LIN {X 0,Y 81.103,Z 363.12,A -85,B 0,C 180,E1 -27834.313,E2 -27834.313} C_VEL
LIN {X 0,Y 82.768,Z 358.459,A -85,B 0,C 180,E1 -27837.848,E2 -27837.848} C_VEL
LIN {X 0,Y 84.322,Z 351.512,A -85,B 0,C 180,E1 -27842.351,E2 -27842.351} C_VEL
LIN {X 0,Y 85.789,Z 343.802,A -85,B 0,C 180,E1 -27846.444,E2 -27846.444} C_VEL
LIN {X 0,Y 86.709,Z 336.677,A -85,B 0,C 180,E1 -27849.672,E2 -27849.672} C_VEL
LIN {X 0,Y 87.275,Z 327.984,A -85,B 0,C 180,E1 -27853.08,E2 -27853.08} C_VEL
LIN {X 0,Y 87.272,Z 324.602,A -85,B 0,C 180,E1 -27854.371,E2 -27854.371} C_VEL
LIN {X 0,Y 84.695,Z 316.637,A -85,B 0,C 180,E1 -27858.324,E2 -27858.324} C_VEL
LIN {X 0,Y 82.109,Z 312.261,A -85,B 0,C 180,E1 -27861.198,E2 -27861.198} C_VEL
LIN {X 0,Y 79.987,Z 309.343,A -85,B 0,C 180,E1 -27863.483,E2 -27863.483} C_VEL
LIN {X 0,Y 79.503,Z 307.393,A -85,B 0,C 180,E1 -27864.498,E2 -27864.498} C_VEL
LIN {X 0,Y 79.529,Z 307.39,A -85,B 0,C 180,E1 -27873.768,E2 -27873.768} C_VEL
LIN {X 0,Y 79.498,Z 307.382,A -85,B 0,C 180,E1 -27879.282,E2 -27879.282} C_VEL
LIN {X 0,Y 79.799,Z 307.348,A -85,B 0,C 180,E1 -27885.672,E2 -27885.672} C_VEL
LIN {X 0,Y 79.947,Z 307.327,A -85,B 0,C 180,E1 -27889.865,E2 -27889.865} C_VEL
LIN {X 0,Y 80.641,Z 307.236,A -85,B 0,C 180,E1 -27899.991,E2 -27899.991} C_VEL
LIN {X 0,Y 80,Z 307.314,A -85,B 0,C 180,E1 -27910.11,E2 -27910.11} C_VEL
LIN {X 0,Y 79.768,Z 307.361,A -85,B 0,C 180,E1 -27915.317,E2 -27915.317} C_VEL
LIN {X 0,Y 79.517,Z 307.376,A -85,B 0,C 180,E1 -27920.693,E2 -27920.693} C_VEL
LIN {X 0,Y 79.487,Z 307.396,A -85,B 0,C 180,E1 -27927.837,E2 -27927.837} C_VEL
LIN {X 0,Y 79.465,Z 307.398,A -85,B 0,C 180,E1 -27937.243,E2 -27937.243} C_VEL
LIN {X 0,Y 79.492,Z 307.392,A -85,B 0,C 180,E1 -27945.001,E2 -27945.001} C_VEL
LIN {X 0,Y 79.475,Z 307.522,A -85,B 0,C 180,E1 -27951.107,E2 -27951.107} C_VEL
LIN {X 0,Y 80.071,Z 309.557,A -85,B 0,C 180,E1 -27952.164,E2 -27952.164} C_VEL
LIN {X 0,Y 81.96,Z 312.404,A -85,B 0,C 180,E1 -27954.533,E2 -27954.533} C_VEL
LIN {X 0,Y 84.975,Z 318.525,A -85,B 0,C 180,E1 -27958.565,E2 -27958.565} C_VEL
LIN {X 0,Y 87.806,Z 325.654,A -85,B 0,C 180,E1 -27962.905,E2 -27962.905} C_VEL
LIN {X 0,Y 89.004,Z 331.434,A -85,B 0,C 180,E1 -27966.098,E2 -27966.098} C_VEL
LIN {X 0,Y 88.877,Z 336.304,A -85,B 0,C 180,E1 -27968.542,E2 -27968.542} C_VEL
LIN {X 0,Y 88.422,Z 338.689,A -85,B 0,C 180,E1 -27969.645,E2 -27969.645} C_VEL
LIN {X 0,Y 84.98,Z 348.04,A -85,B 0,C 180,E1 -27974.402,E2 -27974.402} C_VEL
LIN {X 0,Y 82.427,Z 354.664,A -85,B 0,C 180,E1 -27978.933,E2 -27978.933} C_VEL
LIN {X 0,Y 80.368,Z 360.174,A -85,B 0,C 180,E1 -27983.718,E2 -27983.718} C_VEL
LIN {X 0,Y 78.415,Z 365.767,A -85,B 0,C 180,E1 -27989.993,E2 -27989.993} C_VEL
LIN {X 0,Y 78.325,Z 366.053,A -85,B 0,C 180,E1 -27990.371,E2 -27990.371} C_VEL
LIN {X 0,Y 76.885,Z 368.828,A -85,B 0,C 180,E1 -27994.107,E2 -27994.107} C_VEL
LIN {X 0,Y 73.232,Z 372.559,A -85,B 0,C 180,E1 -28000.555,E2 -28000.555} C_VEL
LIN {X 0,Y 70.419,Z 375.498,A -85,B 0,C 180,E1 -28007.834,E2 -28007.834} C_VEL
LIN {X 0,Y 70.359,Z 376.852,A -85,B 0,C 180,E1 -28012.526,E2 -28012.526} C_VEL
LIN {X 0,Y 71.985,Z 378.249,A -85,B 0,C 180,E1 -28019.211,E2 -28019.211} C_VEL
LIN {X 0,Y 74.077,Z 378.865,A -85,B 0,C 180,E1 -28024.689,E2 -28024.689} C_VEL
LIN {X 0,Y 76.782,Z 378.987,A -85,B 0,C 180,E1 -28029.837,E2 -28029.837} C_VEL
LIN {X 0,Y 81.363,Z 378.263,A -85,B 0,C 180,E1 -28036.302,E2 -28036.302} C_VEL
LIN {X 0,Y 83.749,Z 377.668,A -85,B 0,C 180,E1 -28039.038,E2 -28039.038} C_VEL
LIN {X 0,Y 90.093,Z 375.178,A -85,B 0,C 180,E1 -28044.982,E2 -28044.982} C_VEL
LIN {X 0,Y 97.253,Z 371.306,A -85,B 0,C 180,E1 -28050.121,E2 -28050.121} C_VEL
LIN {X 0,Y 99.807,Z 369.765,A -85,B 0,C 180,E1 -28051.654,E2 -28051.654} C_VEL
LIN {X 0,Y 101.693,Z 367.889,A -85,B 0,C 180,E1 -28053.94,E2 -28053.94} C_VEL
LIN {X 0,Y 102.888,Z 365.535,A -85,B 0,C 180,E1 -28057.941,E2 -28057.941} C_VEL
LIN {X 0,Y 103.573,Z 363.322,A -85,B 0,C 180,E1 -28061.783,E2 -28061.783} C_VEL
LIN {X 0,Y 103.925,Z 362.042,A -85,B 0,C 180,E1 -28064.313,E2 -28064.313} C_VEL
LIN {X 0,Y 104.24,Z 360.271,A -85,B 0,C 180,E1 -28068.338,E2 -28068.338} C_VEL
LIN {X 0,Y 104.447,Z 358.742,A -85,B 0,C 180,E1 -28072.273,E2 -28072.273} C_VEL
LIN {X 0,Y 105.03,Z 356.721,A -85,B 0,C 180,E1 -28080.007,E2 -28080.007} C_VEL
LIN {X 0,Y 105.33,Z 356.2,A -85,B 0,C 180,E1 -28083.833,E2 -28083.833} C_VEL
LIN {X 0,Y 104.851,Z 356.834,A -85,B 0,C 180,E1 -28087.711,E2 -28087.711} C_VEL
LIN {X 0,Y 104.027,Z 359.222,A -85,B 0,C 180,E1 -28095.685,E2 -28095.685} C_VEL
LIN {X 0,Y 103.777,Z 360.902,A -85,B 0,C 180,E1 -28099.799,E2 -28099.799} C_VEL
LIN {X 0,Y 103.283,Z 364.111,A -85,B 0,C 180,E1 -28105.717,E2 -28105.717} C_VEL
LIN {X 0,Y 102.359,Z 367.453,A -85,B 0,C 180,E1 -28111.002,E2 -28111.002} C_VEL
LIN {X 0,Y 101.72,Z 369.604,A -85,B 0,C 180,E1 -28114.004,E2 -28114.004} C_VEL
LIN {X 0,Y 100.581,Z 371.544,A -85,B 0,C 180,E1 -28116.539,E2 -28116.539} C_VEL
LIN {X 0,Y 96.125,Z 375.798,A -85,B 0,C 180,E1 -28121.158,E2 -28121.158} C_VEL
LIN {X 0,Y 92.817,Z 378.218,A -85,B 0,C 180,E1 -28124.01,E2 -28124.01} C_VEL
LIN {X 0,Y 86.169,Z 381.587,A -85,B 0,C 180,E1 -28129.279,E2 -28129.279} C_VEL
LIN {X 0,Y 82.146,Z 383.226,A -85,B 0,C 180,E1 -28133.219,E2 -28133.219} C_VEL
LIN {X 0,Y 78.577,Z 384.271,A -85,B 0,C 180,E1 -28137.552,E2 -28137.552} C_VEL
LIN {X 0,Y 75.641,Z 384.853,A -85,B 0,C 180,E1 -28142.326,E2 -28142.326} C_VEL
LIN {X 0,Y 73.297,Z 385,A -85,B 0,C 180,E1 -28147.455,E2 -28147.455} C_VEL
LIN {X 0,Y 71.542,Z 384.699,A -85,B 0,C 180,E1 -28152.868,E2 -28152.868} C_VEL
LIN {X 0,Y 70.469,Z 383.825,A -85,B 0,C 180,E1 -28158.502,E2 -28158.502} C_VEL
LIN {X 0,Y 70.06,Z 382.441,A -85,B 0,C 180,E1 -28164.25,E2 -28164.25} C_VEL
LIN {X 0,Y 70.143,Z 380.555,A -85,B 0,C 180,E1 -28170.007,E2 -28170.007} C_VEL
LIN {X 0,Y 70.183,Z 376.533,A -85,B 0,C 180,E1 -28178.646,E2 -28178.646} C_VEL
LIN {X 0,Y 70.879,Z 372.999,A -85,B 0,C 180,E1 -28184.36,E2 -28184.36} C_VEL
LIN {X 0,Y 72.632,Z 367.54,A -85,B 0,C 180,E1 -28191.283,E2 -28191.283} C_VEL
LIN {X 0,Y 75.263,Z 360.701,A -85,B 0,C 180,E1 -28197.841,E2 -28197.841} C_VEL
LIN {X 0,Y 77.339,Z 353.736,A -85,B 0,C 180,E1 -28203.049,E2 -28203.049} C_VEL
LIN {X 0,Y 79.321,Z 344.848,A -85,B 0,C 180,E1 -28208.34,E2 -28208.34} C_VEL
LIN {X 0,Y 80.625,Z 336.415,A -85,B 0,C 180,E1 -28212.506,E2 -28212.506} C_VEL
LIN {X 0,Y 81.34,Z 329.032,A -85,B 0,C 180,E1 -28215.661,E2 -28215.661} C_VEL
LIN {X 0,Y 81.384,Z 327.475,A -85,B 0,C 180,E1 -28216.292,E2 -28216.292} C_VEL
LIN {X 0,Y 79.775,Z 321.356,A -85,B 0,C 180,E1 -28219.762,E2 -28219.762} C_VEL
LIN {X 0,Y 75.378,Z 313.535,A -85,B 0,C 180,E1 -28225.974,E2 -28225.974} C_VEL
LIN {X 0,Y 72.881,Z 310.248,A -85,B 0,C 180,E1 -28229.373,E2 -28229.373} C_VEL
LIN {X 0,Y 72.367,Z 308.273,A -85,B 0,C 180,E1 -28230.74,E2 -28230.74} C_VEL
LIN {X 0,Y 72.388,Z 308.265,A -85,B 0,C 180,E1 -28237.138,E2 -28237.138} C_VEL
LIN {X 0,Y 72.69,Z 308.235,A -85,B 0,C 180,E1 -28245.231,E2 -28245.231} C_VEL
LIN {X 0,Y 72.838,Z 308.207,A -85,B 0,C 180,E1 -28248.864,E2 -28248.864} C_VEL
LIN {X 0,Y 73.568,Z 308.116,A -85,B 0,C 180,E1 -28259.99,E2 -28259.99} C_VEL
LIN {X 0,Y 72.886,Z 308.2,A -85,B 0,C 180,E1 -28271.109,E2 -28271.109} C_VEL
LIN {X 0,Y 72.587,Z 308.255,A -85,B 0,C 180,E1 -28276.875,E2 -28276.875} C_VEL
LIN {X 0,Y 72.398,Z 308.262,A -85,B 0,C 180,E1 -28282.837,E2 -28282.837} C_VEL
LIN {X 0,Y 72.378,Z 308.279,A -85,B 0,C 180,E1 -28289.07,E2 -28289.07} C_VEL
LIN {X 0,Y 72.348,Z 308.281,A -85,B 0,C 180,E1 -28295.638,E2 -28295.638} C_VEL
LIN {X 0,Y 72.329,Z 308.288,A -85,B 0,C 180,E1 -28302.842,E2 -28302.842} C_VEL
LIN {X 0,Y 72.465,Z 308.387,A -85,B 0,C 180,E1 -28305.068,E2 -28305.068} C_VEL
LIN {X 0,Y 72.973,Z 310.272,A -85,B 0,C 180,E1 -28306.294,E2 -28306.294} C_VEL
LIN {X 0,Y 75.152,Z 313.541,A -85,B 0,C 180,E1 -28309.756,E2 -28309.756} C_VEL
LIN {X 0,Y 77.952,Z 318.904,A -85,B 0,C 180,E1 -28314.218,E2 -28314.218} C_VEL
LIN {X 0,Y 81.181,Z 326.703,A -85,B 0,C 180,E1 -28319.945,E2 -28319.945} C_VEL
LIN {X 0,Y 82.523,Z 331.958,A -85,B 0,C 180,E1 -28323.382,E2 -28323.382} C_VEL
LIN {X 0,Y 82.753,Z 335.584,A -85,B 0,C 180,E1 -28325.536,E2 -28325.536} C_VEL
LIN {X 0,Y 82.192,Z 339.102,A -85,B 0,C 180,E1 -28327.363,E2 -28327.363} C_VEL
LIN {X 0,Y 78.825,Z 347.551,A -85,B 0,C 180,E1 -28331.81,E2 -28331.81} C_VEL
LIN {X 0,Y 75.411,Z 355.758,A -85,B 0,C 180,E1 -28337.889,E2 -28337.889} C_VEL
LIN {X 0,Y 73.223,Z 361.141,A -85,B 0,C 180,E1 -28343.102,E2 -28343.102} C_VEL
LIN {X 0,Y 71.344,Z 366.236,A -85,B 0,C 180,E1 -28349.444,E2 -28349.444} C_VEL
LIN {X 0,Y 70.153,Z 370.18,A -85,B 0,C 180,E1 -28355.742,E2 -28355.742} C_VEL
LIN {X 0,Y 69.606,Z 374.297,A -85,B 0,C 180,E1 -28364.613,E2 -28364.613} C_VEL
LIN {X 0,Y 70.359,Z 376.852,A -85,B 0,C 180,E1 -28372.526,E2 -28372.526} C_VEL
LIN {X 0,Y 70.741,Z 377.994,A -85,B 0,C 180,E1 -28377.215,E2 -28377.215} C_VEL
LIN {X 0,Y 70.592,Z 379.038,A -85,B 0,C 180,E1 -28385.209,E2 -28385.209} C_VEL
LIN {X 0,Y 71.757,Z 379.279,A -85,B 0,C 180,E1 -28393.169,E2 -28393.169} C_VEL
LIN {X 0,Y 74.073,Z 378.93,A -85,B 0,C 180,E1 -28397.453,E2 -28397.453} C_VEL
LIN {X 0,Y 79.102,Z 377.841,A -85,B 0,C 180,E1 -28403.083,E2 -28403.083} C_VEL
LIN {X 0,Y 86.063,Z 375.201,A -85,B 0,C 180,E1 -28409.018,E2 -28409.018} C_VEL
LIN {X 0,Y 91.133,Z 372.776,A -85,B 0,C 180,E1 -28412.448,E2 -28412.448} C_VEL
LIN {X 0,Y 93.808,Z 371.228,A -85,B 0,C 180,E1 -28414.017,E2 -28414.017} C_VEL
LIN {X 0,Y 95.899,Z 369.544,A -85,B 0,C 180,E1 -28416.583,E2 -28416.583} C_VEL
LIN {X 0,Y 96.958,Z 367.597,A -85,B 0,C 180,E1 -28420.425,E2 -28420.425} C_VEL
LIN {X 0,Y 97.577,Z 366.357,A -85,B 0,C 180,E1 -28423.264,E2 -28423.264} C_VEL
LIN {X 0,Y 98.135,Z 364.597,A -85,B 0,C 180,E1 -28427.601,E2 -28427.601} C_VEL
LIN {X 0,Y 98.601,Z 363.162,A -85,B 0,C 180,E1 -28431.812,E2 -28431.812} C_VEL
LIN {X 0,Y 98.977,Z 362.135,A -85,B 0,C 180,E1 -28435.936,E2 -28435.936} C_VEL
LIN {X 0,Y 99.472,Z 361.225,A -85,B 0,C 180,E1 -28440.007,E2 -28440.007} C_VEL
LIN {X 0,Y 99.771,Z 360.797,A -85,B 0,C 180,E1 -28444.047,E2 -28444.047} C_VEL
LIN {X 0,Y 99.209,Z 361.498,A -85,B 0,C 180,E1 -28448.152,E2 -28448.152} C_VEL
LIN {X 0,Y 98.286,Z 363.955,A -85,B 0,C 180,E1 -28456.627,E2 -28456.627} C_VEL
LIN {X 0,Y 97.745,Z 365.713,A -85,B 0,C 180,E1 -28461.077,E2 -28461.077} C_VEL
LIN {X 0,Y 97.072,Z 368.008,A -85,B 0,C 180,E1 -28465.755,E2 -28465.755} C_VEL
LIN {X 0,Y 95.885,Z 370.907,A -85,B 0,C 180,E1 -28470.877,E2 -28470.877} C_VEL
LIN {X 0,Y 95.224,Z 372.222,A -85,B 0,C 180,E1 -28473.072,E2 -28473.072} C_VEL
LIN {X 0,Y 94.194,Z 373.557,A -85,B 0,C 180,E1 -28474.852,E2 -28474.852} C_VEL
LIN {X 0,Y 90.193,Z 376.729,A -85,B 0,C 180,E1 -28478.821,E2 -28478.821} C_VEL
LIN {X 0,Y 87.979,Z 378.178,A -85,B 0,C 180,E1 -28480.644,E2 -28480.644} C_VEL
LIN {X 0,Y 80.906,Z 381.44,A -85,B 0,C 180,E1 -28485.988,E2 -28485.988} C_VEL
LIN {X 0,Y 76.576,Z 383.034,A -85,B 0,C 180,E1 -28490.035,E2 -28490.035} C_VEL
LIN {X 0,Y 72.682,Z 384.05,A -85,B 0,C 180,E1 -28494.547,E2 -28494.547} C_VEL
LIN {X 0,Y 69.407,Z 384.559,A -85,B 0,C 180,E1 -28499.592,E2 -28499.592} C_VEL
LIN {X 0,Y 66.773,Z 384.631,A -85,B 0,C 180,E1 -28505.111,E2 -28505.111} C_VEL
LIN {X 0,Y 64.779,Z 384.266,A -85,B 0,C 180,E1 -28511.014,E2 -28511.014} C_VEL
LIN {X 0,Y 63.527,Z 383.382,A -85,B 0,C 180,E1 -28517.225,E2 -28517.225} C_VEL
LIN {X 0,Y 63.022,Z 381.928,A -85,B 0,C 180,E1 -28523.606,E2 -28523.606} C_VEL
LIN {X 0,Y 63.059,Z 379.963,A -85,B 0,C 180,E1 -28530.008,E2 -28530.008} C_VEL
LIN {X 0,Y 62.99,Z 377.38,A -85,B 0,C 180,E1 -28536.414,E2 -28536.414} C_VEL
LIN {X 0,Y 63.997,Z 372.229,A -85,B 0,C 180,E1 -28545.943,E2 -28545.943} C_VEL
LIN {X 0,Y 66.032,Z 366.67,A -85,B 0,C 180,E1 -28553.532,E2 -28553.532} C_VEL
LIN {X 0,Y 68.998,Z 359.659,A -85,B 0,C 180,E1 -28560.625,E2 -28560.625} C_VEL
LIN {X 0,Y 71.216,Z 352.438,A -85,B 0,C 180,E1 -28566.316,E2 -28566.316} C_VEL
LIN {X 0,Y 73.153,Z 345.059,A -85,B 0,C 180,E1 -28571.024,E2 -28571.024} C_VEL
LIN {X 0,Y 74.688,Z 336.867,A -85,B 0,C 180,E1 -28575.436,E2 -28575.436} C_VEL
LIN {X 0,Y 75.561,Z 329.807,A -85,B 0,C 180,E1 -28578.792,E2 -28578.792} C_VEL
LIN {X 0,Y 74.909,Z 326.782,A -85,B 0,C 180,E1 -28580.695,E2 -28580.695} C_VEL
LIN {X 0,Y 72.798,Z 322.258,A -85,B 0,C 180,E1 -28584.591,E2 -28584.591} C_VEL
LIN {X 0,Y 70.569,Z 318.168,A -85,B 0,C 180,E1 -28588.465,E2 -28588.465} C_VEL
LIN {X 0,Y 68.016,Z 313.925,A -85,B 0,C 180,E1 -28593.379,E2 -28593.379} C_VEL
LIN {X 0,Y 66.142,Z 311.65,A -85,B 0,C 180,E1 -28596.921,E2 -28596.921} C_VEL
LIN {X 0,Y 65.314,Z 309.148,A -85,B 0,C 180,E1 -28599.519,E2 -28599.519} C_VEL
LIN {X 0,Y 65.732,Z 309.091,A -85,B 0,C 180,E1 -28607.642,E2 -28607.642} C_VEL
LIN {X 0,Y 66.466,Z 309,A -85,B 0,C 180,E1 -28619.989,E2 -28619.989} C_VEL
LIN {X 0,Y 65.942,Z 309.081,A -85,B 0,C 180,E1 -28626.107,E2 -28626.107} C_VEL
LIN {X 0,Y 65.779,Z 309.088,A -85,B 0,C 180,E1 -28632.327,E2 -28632.327} C_VEL
LIN {X 0,Y 65.39,Z 309.144,A -85,B 0,C 180,E1 -28638.798,E2 -28638.798} C_VEL
LIN {X 0,Y 65.25,Z 309.165,A -85,B 0,C 180,E1 -28645.508,E2 -28645.508} C_VEL
LIN {X 0,Y 65.221,Z 309.174,A -85,B 0,C 180,E1 -28652.587,E2 -28652.587} C_VEL
LIN {X 0,Y 65.334,Z 309.367,A -85,B 0,C 180,E1 -28656.259,E2 -28656.259} C_VEL
LIN {X 0,Y 65.799,Z 311.001,A -85,B 0,C 180,E1 -28657.876,E2 -28657.876} C_VEL
LIN {X 0,Y 67.783,Z 313.741,A -85,B 0,C 180,E1 -28662.229,E2 -28662.229} C_VEL
LIN {X 0,Y 70.259,Z 317.764,A -85,B 0,C 180,E1 -28667.066,E2 -28667.066} C_VEL
LIN {X 0,Y 72.915,Z 323.466,A -85,B 0,C 180,E1 -28672.657,E2 -28672.657} C_VEL
LIN {X 0,Y 75.017,Z 329.123,A -85,B 0,C 180,E1 -28677.457,E2 -28677.457} C_VEL
LIN {X 0,Y 76.285,Z 333.805,A -85,B 0,C 180,E1 -28681.009,E2 -28681.009} C_VEL
LIN {X 0,Y 76.509,Z 337.183,A -85,B 0,C 180,E1 -28683.389,E2 -28683.389} C_VEL
LIN {X 0,Y 76.114,Z 339.515,A -85,B 0,C 180,E1 -28684.712,E2 -28684.712} C_VEL
LIN {X 0,Y 72.108,Z 348.813,A -85,B 0,C 180,E1 -28690.047,E2 -28690.047} C_VEL
LIN {X 0,Y 69.111,Z 355.415,A -85,B 0,C 180,E1 -28695.264,E2 -28695.264} C_VEL
LIN {X 0,Y 66.658,Z 360.911,A -85,B 0,C 180,E1 -28700.893,E2 -28700.893} C_VEL
LIN {X 0,Y 64.705,Z 365.52,A -85,B 0,C 180,E1 -28706.879,E2 -28706.879} C_VEL
LIN {X 0,Y 63.357,Z 369.531,A -85,B 0,C 180,E1 -28713.509,E2 -28713.509} C_VEL
LIN {X 0,Y 62.52,Z 373.752,A -85,B 0,C 180,E1 -28722.984,E2 -28722.984} C_VEL
LIN {X 0,Y 62.803,Z 375.992,A -85,B 0,C 180,E1 -28729.607,E2 -28729.607} C_VEL
LIN {X 0,Y 63.892,Z 377.664,A -85,B 0,C 180,E1 -28736.094,E2 -28736.094} C_VEL
LIN {X 0,Y 65.667,Z 378.723,A -85,B 0,C 180,E1 -28742.342,E2 -28742.342} C_VEL
LIN {X 0,Y 68.155,Z 379.251,A -85,B 0,C 180,E1 -28748.212,E2 -28748.212} C_VEL
LIN {X 0,Y 71.301,Z 379.283,A -85,B 0,C 180,E1 -28753.617,E2 -28753.617} C_VEL
LIN {X 0,Y 74.073,Z 378.93,A -85,B 0,C 180,E1 -28757.453,E2 -28757.453} C_VEL
LIN {X 0,Y 76.749,Z 378.431,A -85,B 0,C 180,E1 -28761.441,E2 -28761.441} C_VEL
LIN {X 0,Y 80.34,Z 376.992,A -85,B 0,C 180,E1 -28768.109,E2 -28768.109} C_VEL
LIN {X 0,Y 84.66,Z 374.573,A -85,B 0,C 180,E1 -28774.095,E2 -28774.095} C_VEL
LIN {X 0,Y 88.275,Z 372.535,A -85,B 0,C 180,E1 -28776.894,E2 -28776.894} C_VEL
LIN {X 0,Y 90.057,Z 371.146,A -85,B 0,C 180,E1 -28779.45,E2 -28779.45} C_VEL
LIN {X 0,Y 90.785,Z 370.22,A -85,B 0,C 180,E1 -28781.97,E2 -28781.97} C_VEL
LIN {X 0,Y 91.685,Z 368.508,A -85,B 0,C 180,E1 -28786.714,E2 -28786.714} C_VEL
LIN {X 0,Y 92.427,Z 367.193,A -85,B 0,C 180,E1 -28791.261,E2 -28791.261} C_VEL
LIN {X 0,Y 93,Z 366.154,A -85,B 0,C 180,E1 -28795.674,E2 -28795.674} C_VEL
LIN {X 0,Y 93.575,Z 365.328,A -85,B 0,C 180,E1 -28800.008,E2 -28800.008} C_VEL
LIN {X 0,Y 93.902,Z 365.023,A -85,B 0,C 180,E1 -28804.3,E2 -28804.3} C_VEL
LIN {X 0,Y 92.931,Z 366.213,A -85,B 0,C 180,E1 -28810.57,E2 -28810.57} C_VEL
LIN {X 0,Y 92.023,Z 368.332,A -85,B 0,C 180,E1 -28817.795,E2 -28817.795} C_VEL
LIN {X 0,Y 91.252,Z 370.118,A -85,B 0,C 180,E1 -28822.657,E2 -28822.657} C_VEL
LIN {X 0,Y 90.04,Z 372.537,A -85,B 0,C 180,E1 -28827.934,E2 -28827.934} C_VEL
LIN {X 0,Y 89.377,Z 373.689,A -85,B 0,C 180,E1 -28830.134,E2 -28830.134} C_VEL
LIN {X 0,Y 87.87,Z 375.231,A -85,B 0,C 180,E1 -28832.892,E2 -28832.892} C_VEL
LIN {X 0,Y 85.533,Z 376.888,A -85,B 0,C 180,E1 -28835.121,E2 -28835.121} C_VEL
LIN {X 0,Y 83.342,Z 378.166,A -85,B 0,C 180,E1 -28836.953,E2 -28836.953} C_VEL
LIN {X 0,Y 75.947,Z 381.294,A -85,B 0,C 180,E1 -28842.253,E2 -28842.253} C_VEL
LIN {X 0,Y 71.28,Z 382.818,A -85,B 0,C 180,E1 -28846.366,E2 -28846.366} C_VEL
LIN {X 0,Y 67.025,Z 383.824,A -85,B 0,C 180,E1 -28851.024,E2 -28851.024} C_VEL
LIN {X 0,Y 63.365,Z 384.264,A -85,B 0,C 180,E1 -28856.329,E2 -28856.329} C_VEL
LIN {X 0,Y 60.391,Z 384.264,A -85,B 0,C 180,E1 -28862.268,E2 -28862.268} C_VEL
LIN {X 0,Y 58.107,Z 383.825,A -85,B 0,C 180,E1 -28868.735,E2 -28868.735} C_VEL
LIN {X 0,Y 56.614,Z 382.916,A -85,B 0,C 180,E1 -28875.634,E2 -28875.634} C_VEL
LIN {X 0,Y 55.889,Z 380.484,A -85,B 0,C 180,E1 -28886.405,E2 -28886.405} C_VEL
LIN {X 0,Y 55.977,Z 379.372,A -85,B 0,C 180,E1 -28890.009,E2 -28890.009} C_VEL
LIN {X 0,Y 55.933,Z 376.703,A -85,B 0,C 180,E1 -28897.228,E2 -28897.228} C_VEL
LIN {X 0,Y 56.587,Z 373.391,A -85,B 0,C 180,E1 -28904.392,E2 -28904.392} C_VEL
LIN {X 0,Y 58.437,Z 368.164,A -85,B 0,C 180,E1 -28913.018,E2 -28913.018} C_VEL
LIN {X 0,Y 60.784,Z 363.037,A -85,B 0,C 180,E1 -28919.442,E2 -28919.442} C_VEL
LIN {X 0,Y 62.874,Z 358.546,A -85,B 0,C 180,E1 -28923.989,E2 -28923.989} C_VEL
LIN {X 0,Y 65.375,Z 351.116,A -85,B 0,C 180,E1 -28930.177,E2 -28930.177} C_VEL
LIN {X 0,Y 67.453,Z 343.961,A -85,B 0,C 180,E1 -28935.006,E2 -28935.006} C_VEL
LIN {X 0,Y 69.198,Z 336.038,A -85,B 0,C 180,E1 -28939.531,E2 -28939.531} C_VEL
LIN {X 0,Y 69.774,Z 332.099,A -85,B 0,C 180,E1 -28941.678,E2 -28941.678} C_VEL
LIN {X 0,Y 68.903,Z 329.013,A -85,B 0,C 180,E1 -28944.258,E2 -28944.258} C_VEL
LIN {X 0,Y 66.459,Z 323.752,A -85,B 0,C 180,E1 -28949.835,E2 -28949.835} C_VEL
LIN {X 0,Y 64.589,Z 320.325,A -85,B 0,C 180,E1 -28954.188,E2 -28954.188} C_VEL
LIN {X 0,Y 62.717,Z 317.648,A -85,B 0,C 180,E1 -28958.63,E2 -28958.63} C_VEL
LIN {X 0,Y 62.276,Z 316.478,A -85,B 0,C 180,E1 -28960.199,E2 -28960.199} C_VEL
LIN {X 0,Y 61.209,Z 314.774,A -85,B 0,C 180,E1 -28963.548,E2 -28963.548} C_VEL
LIN {X 0,Y 59.096,Z 311.463,A -85,B 0,C 180,E1 -28972.084,E2 -28972.084} C_VEL
LIN {X 0,Y 58.918,Z 309.955,A -85,B 0,C 180,E1 -28974.855,E2 -28974.855} C_VEL
LIN {X 0,Y 59.359,Z 309.884,A -85,B 0,C 180,E1 -28979.988,E2 -28979.988} C_VEL
LIN {X 0,Y 58.825,Z 309.963,A -85,B 0,C 180,E1 -28986.849,E2 -28986.849} C_VEL
LIN {X 0,Y 58.531,Z 310.007,A -85,B 0,C 180,E1 -28996.109,E2 -28996.109} C_VEL
LIN {X 0,Y 58.352,Z 310.251,A -85,B 0,C 180,E1 -28998.938,E2 -28998.938} C_VEL
LIN {X 0,Y 58.498,Z 311.356,A -85,B 0,C 180,E1 -29001.112,E2 -29001.112} C_VEL
LIN {X 0,Y 61.911,Z 315.674,A -85,B 0,C 180,E1 -29014.567,E2 -29014.567} C_VEL
LIN {X 0,Y 63.327,Z 318.61,A -85,B 0,C 180,E1 -29019.014,E2 -29019.014} C_VEL
LIN {X 0,Y 65.406,Z 322.274,A -85,B 0,C 180,E1 -29024.543,E2 -29024.543} C_VEL
LIN {X 0,Y 67.85,Z 327.946,A -85,B 0,C 180,E1 -29030.96,E2 -29030.96} C_VEL
LIN {X 0,Y 69.62,Z 333.57,A -85,B 0,C 180,E1 -29036.369,E2 -29036.369} C_VEL
LIN {X 0,Y 70.347,Z 337.695,A -85,B 0,C 180,E1 -29040.023,E2 -29040.023} C_VEL
LIN {X 0,Y 70.207,Z 339.934,A -85,B 0,C 180,E1 -29041.6,E2 -29041.6} C_VEL
LIN {X 0,Y 66.288,Z 348.331,A -85,B 0,C 180,E1 -29046.564,E2 -29046.564} C_VEL
LIN {X 0,Y 62.21,Z 356.51,A -85,B 0,C 180,E1 -29053.586,E2 -29053.586} C_VEL
LIN {X 0,Y 59.564,Z 361.879,A -85,B 0,C 180,E1 -29059.797,E2 -29059.797} C_VEL
LIN {X 0,Y 57.533,Z 366.37,A -85,B 0,C 180,E1 -29066.489,E2 -29066.489} C_VEL
LIN {X 0,Y 56.282,Z 369.822,A -85,B 0,C 180,E1 -29072.902,E2 -29072.902} C_VEL
LIN {X 0,Y 55.476,Z 373.198,A -85,B 0,C 180,E1 -29080.945,E2 -29080.945} C_VEL
LIN {X 0,Y 55.981,Z 376.552,A -85,B 0,C 180,E1 -29092.115,E2 -29092.115} C_VEL
LIN {X 0,Y 58.326,Z 378.638,A -85,B 0,C 180,E1 -29102.516,E2 -29102.516} C_VEL
LIN {X 0,Y 59.584,Z 379.194,A -85,B 0,C 180,E1 -29106.128,E2 -29106.128} C_VEL
LIN {X 0,Y 62.557,Z 379.636,A -85,B 0,C 180,E1 -29112.371,E2 -29112.371} C_VEL
LIN {X 0,Y 68.143,Z 379.31,A -85,B 0,C 180,E1 -29120.582,E2 -29120.582} C_VEL
LIN {X 0,Y 74.907,Z 377.976,A -85,B 0,C 180,E1 -29127.594,E2 -29127.594} C_VEL
LIN {X 0,Y 82.506,Z 375.23,A -85,B 0,C 180,E1 -29133.417,E2 -29133.417} C_VEL
LIN {X 0,Y 88.275,Z 372.535,A -85,B 0,C 180,E1 -29136.894,E2 -29136.894} C_VEL
LIN {X 0,Y 89.7,Z 371.609,A -85,B 0,C 180,E1 -29138.232,E2 -29138.232} C_VEL
LIN {X 0,Y 90.513,Z 370.722,A -85,B 0,C 180,E1 -29140.431,E2 -29140.431} C_VEL
LIN {X 0,Y 90.361,Z 370.059,A -85,B 0,C 180,E1 -29143.478,E2 -29143.478} C_VEL
LIN {X 0,Y 89.654,Z 369.833,A -85,B 0,C 180,E1 -29145.946,E2 -29145.946} C_VEL
LIN {X 0,Y 86.849,Z 369.578,A -85,B 0,C 180,E1 -29156.265,E2 -29156.265} C_VEL
LIN {X 0,Y 86.979,Z 369.387,A -85,B 0,C 180,E1 -29157.77,E2 -29157.77} C_VEL
LIN {X 0,Y 87.414,Z 369.039,A -85,B 0,C 180,E1 -29160.008,E2 -29160.008} C_VEL
LIN {X 0,Y 87.732,Z 368.866,A -85,B 0,C 180,E1 -29164.603,E2 -29164.603} C_VEL
LIN {X 0,Y 86.955,Z 369.631,A -85,B 0,C 180,E1 -29169.311,E2 -29169.311} C_VEL
LIN {X 0,Y 86.125,Z 370.764,A -85,B 0,C 180,E1 -29174.179,E2 -29174.179} C_VEL
LIN {X 0,Y 85.335,Z 372.239,A -85,B 0,C 180,E1 -29179.243,E2 -29179.243} C_VEL
LIN {X 0,Y 84.172,Z 374.12,A -85,B 0,C 180,E1 -29184.684,E2 -29184.684} C_VEL
LIN {X 0,Y 83.368,Z 375.178,A -85,B 0,C 180,E1 -29187.403,E2 -29187.403} C_VEL
LIN {X 0,Y 81.654,Z 376.791,A -85,B 0,C 180,E1 -29190.617,E2 -29190.617} C_VEL
LIN {X 0,Y 76.697,Z 379.23,A -85,B 0,C 180,E1 -29194.454,E2 -29194.454} C_VEL
LIN {X 0,Y 71.354,Z 381.157,A -85,B 0,C 180,E1 -29198.018,E2 -29198.018} C_VEL
LIN {X 0,Y 66.323,Z 382.602,A -85,B 0,C 180,E1 -29202.131,E2 -29202.131} C_VEL
LIN {X 0,Y 61.671,Z 383.574,A -85,B 0,C 180,E1 -29206.874,E2 -29206.874} C_VEL
LIN {X 0,Y 57.572,Z 383.971,A -85,B 0,C 180,E1 -29212.396,E2 -29212.396} C_VEL
LIN {X 0,Y 54.199,Z 383.897,A -85,B 0,C 180,E1 -29218.768,E2 -29218.768} C_VEL
LIN {X 0,Y 51.558,Z 383.385,A -85,B 0,C 180,E1 -29225.873,E2 -29225.873} C_VEL
LIN {X 0,Y 49.77,Z 382.424,A -85,B 0,C 180,E1 -29233.607,E2 -29233.607} C_VEL
LIN {X 0,Y 48.852,Z 379.895,A -85,B 0,C 180,E1 -29245.886,E2 -29245.886} C_VEL
LIN {X 0,Y 48.882,Z 378.78,A -85,B 0,C 180,E1 -29250.011,E2 -29250.011} C_VEL
LIN {X 0,Y 49.189,Z 374.49,A -85,B 0,C 180,E1 -29262.386,E2 -29262.386} C_VEL
LIN {X 0,Y 51.382,Z 368.478,A -85,B 0,C 180,E1 -29274.237,E2 -29274.237} C_VEL
LIN {X 0,Y 53.921,Z 363.485,A -85,B 0,C 180,E1 -29281.434,E2 -29281.434} C_VEL
LIN {X 0,Y 56.946,Z 357.403,A -85,B 0,C 180,E1 -29288.114,E2 -29288.114} C_VEL
LIN {X 0,Y 59.837,Z 349.782,A -85,B 0,C 180,E1 -29294.818,E2 -29294.818} C_VEL
LIN {X 0,Y 62.138,Z 342.767,A -85,B 0,C 180,E1 -29299.779,E2 -29299.779} C_VEL
LIN {X 0,Y 63.979,Z 335.611,A -85,B 0,C 180,E1 -29304.121,E2 -29304.121} C_VEL
LIN {X 0,Y 64.074,Z 334.512,A -85,B 0,C 180,E1 -29304.863,E2 -29304.863} C_VEL
LIN {X 0,Y 62.052,Z 329.176,A -85,B 0,C 180,E1 -29311.213,E2 -29311.213} C_VEL
LIN {X 0,Y 60.468,Z 325.803,A -85,B 0,C 180,E1 -29315.984,E2 -29315.984} C_VEL
LIN {X 0,Y 58.67,Z 322.118,A -85,B 0,C 180,E1 -29322.562,E2 -29322.562} C_VEL
LIN {X 0,Y 56.455,Z 318.229,A -85,B 0,C 180,E1 -29332.836,E2 -29332.836} C_VEL
LIN {X 0,Y 56.264,Z 316.538,A -85,B 0,C 180,E1 -29336.406,E2 -29336.406} C_VEL
LIN {X 0,Y 55.849,Z 316.05,A -85,B 0,C 180,E1 -29339.987,E2 -29339.987} C_VEL
LIN {X 0,Y 55.764,Z 316.644,A -85,B 0,C 180,E1 -29356.932,E2 -29356.932} C_VEL
LIN {X 0,Y 56.608,Z 319.696,A -85,B 0,C 180,E1 -29365.741,E2 -29365.741} C_VEL
LIN {X 0,Y 58.176,Z 321.483,A -85,B 0,C 180,E1 -29372.243,E2 -29372.243} C_VEL
LIN {X 0,Y 60.51,Z 326.454,A -85,B 0,C 180,E1 -29381.209,E2 -29381.209} C_VEL
LIN {X 0,Y 62.651,Z 332.308,A -85,B 0,C 180,E1 -29389.162,E2 -29389.162} C_VEL
LIN {X 0,Y 64.092,Z 338.303,A -85,B 0,C 180,E1 -29395.798,E2 -29395.798} C_VEL
LIN {X 0,Y 64.336,Z 340.409,A -85,B 0,C 180,E1 -29397.813,E2 -29397.813} C_VEL
LIN {X 0,Y 63.449,Z 342.612,A -85,B 0,C 180,E1 -29399.174,E2 -29399.174} C_VEL
LIN {X 0,Y 59.835,Z 349.585,A -85,B 0,C 180,E1 -29403.857,E2 -29403.857} C_VEL
LIN {X 0,Y 56.211,Z 356.168,A -85,B 0,C 180,E1 -29409.88,E2 -29409.88} C_VEL
LIN {X 0,Y 53.192,Z 361.649,A -85,B 0,C 180,E1 -29416.621,E2 -29416.621} C_VEL
LIN {X 0,Y 50.35,Z 367.221,A -85,B 0,C 180,E1 -29425.988,E2 -29425.988} C_VEL
LIN {X 0,Y 48.913,Z 370.864,A -85,B 0,C 180,E1 -29434.104,E2 -29434.104} C_VEL
LIN {X 0,Y 48.409,Z 375.057,A -85,B 0,C 180,E1 -29446.868,E2 -29446.868} C_VEL
LIN {X 0,Y 49.277,Z 377.111,A -85,B 0,C 180,E1 -29455.32,E2 -29455.32} C_VEL
LIN {X 0,Y 51.819,Z 378.93,A -85,B 0,C 180,E1 -29465.561,E2 -29465.561} C_VEL
LIN {X 0,Y 53.828,Z 379.628,A -85,B 0,C 180,E1 -29470.742,E2 -29470.742} C_VEL
LIN {X 0,Y 57.349,Z 380.019,A -85,B 0,C 180,E1 -29477.318,E2 -29477.318} C_VEL
LIN {X 0,Y 61.498,Z 379.879,A -85,B 0,C 180,E1 -29483.111,E2 -29483.111} C_VEL
LIN {X 0,Y 66.146,Z 379.246,A -85,B 0,C 180,E1 -29488.196,E2 -29488.196} C_VEL
LIN {X 0,Y 71.229,Z 378.105,A -85,B 0,C 180,E1 -29492.608,E2 -29492.608} C_VEL
LIN {X 0,Y 76.646,Z 376.425,A -85,B 0,C 180,E1 -29496.465,E2 -29496.465} C_VEL
LIN {X 0,Y 83.176,Z 373.736,A -85,B 0,C 180,E1 -29500.256,E2 -29500.256} C_VEL
LIN {X 0,Y 84.841,Z 371.997,A -85,B 0,C 180,E1 -29505.62,E2 -29505.62} C_VEL
LIN {X 0,Y 85.914,Z 370.781,A -85,B 0,C 180,E1 -29510.592,E2 -29510.592} C_VEL
LIN {X 0,Y 86.663,Z 369.759,A -85,B 0,C 180,E1 -29515.357,E2 -29515.357} C_VEL
LIN {X 0,Y 86.979,Z 369.387,A -85,B 0,C 180,E1 -29517.77,E2 -29517.77} C_VEL
LIN {X 0,Y 86.955,Z 369.294,A -85,B 0,C 180,E1 -29520.325,E2 -29520.325} C_VEL
LIN {X 0,Y 85.737,Z 369.988,A -85,B 0,C 180,E1 -29524.122,E2 -29524.122} C_VEL
LIN {X 0,Y 83.731,Z 371.245,A -85,B 0,C 180,E1 -29527.843,E2 -29527.843} C_VEL
LIN {X 0,Y 79.388,Z 374.26,A -85,B 0,C 180,E1 -29535.937,E2 -29535.937} C_VEL
LIN {X 0,Y 78.567,Z 375.099,A -85,B 0,C 180,E1 -29538.869,E2 -29538.869} C_VEL
LIN {X 0,Y 78.231,Z 375.671,A -85,B 0,C 180,E1 -29541.069,E2 -29541.069} C_VEL
LIN {X 0,Y 77.295,Z 376.799,A -85,B 0,C 180,E1 -29544.616,E2 -29544.616} C_VEL
LIN {X 0,Y 75.79,Z 377.875,A -85,B 0,C 180,E1 -29547.633,E2 -29547.633} C_VEL
LIN {X 0,Y 72.843,Z 379.177,A -85,B 0,C 180,E1 -29549.749,E2 -29549.749} C_VEL
LIN {X 0,Y 67.203,Z 381.021,A -85,B 0,C 180,E1 -29553.229,E2 -29553.229} C_VEL
LIN {X 0,Y 61.787,Z 382.387,A -85,B 0,C 180,E1 -29557.245,E2 -29557.245} C_VEL
LIN {X 0,Y 56.702,Z 383.298,A -85,B 0,C 180,E1 -29561.969,E2 -29561.969} C_VEL
LIN {X 0,Y 52.113,Z 383.678,A -85,B 0,C 180,E1 -29567.614,E2 -29567.614} C_VEL
LIN {X 0,Y 48.264,Z 383.527,A -85,B 0,C 180,E1 -29574.39,E2 -29574.39} C_VEL
LIN {X 0,Y 45.18,Z 382.94,A -85,B 0,C 180,E1 -29582.195,E2 -29582.195} C_VEL
LIN {X 0,Y 43.019,Z 381.904,A -85,B 0,C 180,E1 -29590.942,E2 -29590.942} C_VEL
LIN {X 0,Y 41.797,Z 379.299,A -85,B 0,C 180,E1 -29605.19,E2 -29605.19} C_VEL
LIN {X 0,Y 41.781,Z 378.182,A -85,B 0,C 180,E1 -29610.013,E2 -29610.013} C_VEL
LIN {X 0,Y 42.253,Z 373.76,A -85,B 0,C 180,E1 -29624.461,E2 -29624.461} C_VEL
LIN {X 0,Y 44.343,Z 368.782,A -85,B 0,C 180,E1 -29635.852,E2 -29635.852} C_VEL
LIN {X 0,Y 47.969,Z 362.492,A -85,B 0,C 180,E1 -29645.89,E2 -29645.89} C_VEL
LIN {X 0,Y 50.561,Z 358.006,A -85,B 0,C 180,E1 -29651.333,E2 -29651.333} C_VEL
LIN {X 0,Y 53.514,Z 351.489,A -85,B 0,C 180,E1 -29657.83,E2 -29657.83} C_VEL
LIN {X 0,Y 56.555,Z 343.757,A -85,B 0,C 180,E1 -29663.892,E2 -29663.892} C_VEL
LIN {X 0,Y 58.348,Z 338.446,A -85,B 0,C 180,E1 -29667.49,E2 -29667.49} C_VEL
LIN {X 0,Y 58.257,Z 337.016,A -85,B 0,C 180,E1 -29668.942,E2 -29668.942} C_VEL
LIN {X 0,Y 56.53,Z 332.176,A -85,B 0,C 180,E1 -29676.155,E2 -29676.155} C_VEL
LIN {X 0,Y 54.741,Z 327.545,A -85,B 0,C 180,E1 -29685.108,E2 -29685.108} C_VEL
LIN {X 0,Y 53.21,Z 322.676,A -85,B 0,C 180,E1 -29699.986,E2 -29699.986} C_VEL
LIN {X 0,Y 52.897,Z 323.04,A -85,B 0,C 180,E1 -29715.396,E2 -29715.396} C_VEL
LIN {X 0,Y 53.132,Z 325.512,A -85,B 0,C 180,E1 -29723.364,E2 -29723.364} C_VEL
LIN {X 0,Y 54.534,Z 327.546,A -85,B 0,C 180,E1 -29731.014,E2 -29731.014} C_VEL
LIN {X 0,Y 55.88,Z 331.308,A -85,B 0,C 180,E1 -29738.947,E2 -29738.947} C_VEL
LIN {X 0,Y 57.413,Z 336.634,A -85,B 0,C 180,E1 -29747.242,E2 -29747.242} C_VEL
LIN {X 0,Y 58.187,Z 340.993,A -85,B 0,C 180,E1 -29752.838,E2 -29752.838} C_VEL
LIN {X 0,Y 58.026,Z 342.961,A -85,B 0,C 180,E1 -29754.868,E2 -29754.868} C_VEL
LIN {X 0,Y 53.541,Z 350.784,A -85,B 0,C 180,E1 -29760.501,E2 -29760.501} C_VEL
LIN {X 0,Y 49.545,Z 357.229,A -85,B 0,C 180,E1 -29767.029,E2 -29767.029} C_VEL
LIN {X 0,Y 46.21,Z 362.59,A -85,B 0,C 180,E1 -29774.553,E2 -29774.553} C_VEL
LIN {X 0,Y 43.149,Z 368.05,A -85,B 0,C 180,E1 -29785.317,E2 -29785.317} C_VEL
LIN {X 0,Y 41.675,Z 371.594,A -85,B 0,C 180,E1 -29794.819,E2 -29794.819} C_VEL
LIN {X 0,Y 41.479,Z 375.696,A -85,B 0,C 180,E1 -29809.795,E2 -29809.795} C_VEL
LIN {X 0,Y 42.785,Z 377.661,A -85,B 0,C 180,E1 -29819.51,E2 -29819.51} C_VEL
LIN {X 0,Y 45.506,Z 379.22,A -85,B 0,C 180,E1 -29829.475,E2 -29829.475} C_VEL
LIN {X 0,Y 48.498,Z 380.026,A -85,B 0,C 180,E1 -29836.417,E2 -29836.417} C_VEL
LIN {X 0,Y 52.639,Z 380.398,A -85,B 0,C 180,E1 -29843.216,E2 -29843.216} C_VEL
LIN {X 0,Y 61.042,Z 379.732,A -85,B 0,C 180,E1 -29852.593,E2 -29852.593} C_VEL
LIN {X 0,Y 68.15,Z 378.233,A -85,B 0,C 180,E1 -29858.122,E2 -29858.122} C_VEL
LIN {X 0,Y 74.013,Z 376.469,A -85,B 0,C 180,E1 -29861.7,E2 -29861.7} C_VEL
LIN {X 0,Y 77.398,Z 375.083,A -85,B 0,C 180,E1 -29864.202,E2 -29864.202} C_VEL
LIN {X 0,Y 79.039,Z 373.86,A -85,B 0,C 180,E1 -29869.766,E2 -29869.766} C_VEL
LIN {X 0,Y 80.074,Z 372.94,A -85,B 0,C 180,E1 -29874.974,E2 -29874.974} C_VEL
LIN {X 0,Y 81.02,Z 372.339,A -85,B 0,C 180,E1 -29880.009,E2 -29880.009} C_VEL
LIN {X 0,Y 81.303,Z 372.294,A -85,B 0,C 180,E1 -29884.968,E2 -29884.968} C_VEL
LIN {X 0,Y 80.385,Z 373.066,A -85,B 0,C 180,E1 -29890.079,E2 -29890.079} C_VEL
LIN {X 0,Y 79.337,Z 374.191,A -85,B 0,C 180,E1 -29895.421,E2 -29895.421} C_VEL
LIN {X 0,Y 78.567,Z 375.099,A -85,B 0,C 180,E1 -29898.869,E2 -29898.869} C_VEL
LIN {X 0,Y 77.555,Z 375.96,A -85,B 0,C 180,E1 -29901.089,E2 -29901.089} C_VEL
LIN {X 0,Y 75.078,Z 377.275,A -85,B 0,C 180,E1 -29903.522,E2 -29903.522} C_VEL
LIN {X 0,Y 70.536,Z 379.157,A -85,B 0,C 180,E1 -29906.225,E2 -29906.225} C_VEL
LIN {X 0,Y 64.984,Z 380.794,A -85,B 0,C 180,E1 -29908.623,E2 -29908.623} C_VEL
LIN {X 0,Y 57.205,Z 382.304,A -85,B 0,C 180,E1 -29912.345,E2 -29912.345} C_VEL
LIN {X 0,Y 53.603,Z 382.795,A -85,B 0,C 180,E1 -29914.935,E2 -29914.935} C_VEL
LIN {X 0,Y 47.101,Z 383.367,A -85,B 0,C 180,E1 -29921.767,E2 -29921.767} C_VEL
LIN {X 0,Y 42.692,Z 383.159,A -85,B 0,C 180,E1 -29928.833,E2 -29928.833} C_VEL
LIN {X 0,Y 39.026,Z 382.492,A -85,B 0,C 180,E1 -29937.315,E2 -29937.315} C_VEL
LIN {X 0,Y 36.376,Z 381.378,A -85,B 0,C 180,E1 -29947.285,E2 -29947.285} C_VEL
LIN {X 0,Y 34.992,Z 379.791,A -85,B 0,C 180,E1 -29958.429,E2 -29958.429} C_VEL
LIN {X 0,Y 34.686,Z 377.575,A -85,B 0,C 180,E1 -29970.015,E2 -29970.015} C_VEL
LIN {X 0,Y 35.402,Z 372.977,A -85,B 0,C 180,E1 -29987.34,E2 -29987.34} C_VEL
LIN {X 0,Y 38.067,Z 367.884,A -85,B 0,C 180,E1 -30000.527,E2 -30000.527} C_VEL
LIN {X 0,Y 41.421,Z 362.905,A -85,B 0,C 180,E1 -30009.53,E2 -30009.53} C_VEL
LIN {X 0,Y 44.372,Z 358.547,A -85,B 0,C 180,E1 -30015.476,E2 -30015.476} C_VEL
LIN {X 0,Y 48.74,Z 350.217,A -85,B 0,C 180,E1 -30024.27,E2 -30024.27} C_VEL
LIN {X 0,Y 51.785,Z 343.578,A -85,B 0,C 180,E1 -30029.699,E2 -30029.699} C_VEL
LIN {X 0,Y 52.387,Z 342.022,A -85,B 0,C 180,E1 -30030.829,E2 -30030.829} C_VEL
LIN {X 0,Y 52.684,Z 340.316,A -85,B 0,C 180,E1 -30032.602,E2 -30032.602} C_VEL
LIN {X 0,Y 51.637,Z 336.183,A -85,B 0,C 180,E1 -30040.093,E2 -30040.093} C_VEL
LIN {X 0,Y 50.655,Z 332.967,A -85,B 0,C 180,E1 -30047.567,E2 -30047.567} C_VEL
LIN {X 0,Y 50.018,Z 329.291,A -85,B 0,C 180,E1 -30059.986,E2 -30059.986} C_VEL
LIN {X 0,Y 49.57,Z 329.144,A -85,B 0,C 180,E1 -30068.136,E2 -30068.136} C_VEL
LIN {X 0,Y 49.479,Z 330.083,A -85,B 0,C 180,E1 -30076.488,E2 -30076.488} C_VEL
LIN {X 0,Y 50.401,Z 333.149,A -85,B 0,C 180,E1 -30089.195,E2 -30089.195} C_VEL
LIN {X 0,Y 51.358,Z 336.9,A -85,B 0,C 180,E1 -30097.986,E2 -30097.986} C_VEL
LIN {X 0,Y 51.84,Z 339.375,A -85,B 0,C 180,E1 -30102.656,E2 -30102.656} C_VEL
LIN {X 0,Y 52.267,Z 342.617,A -85,B 0,C 180,E1 -30107.741,E2 -30107.741} C_VEL
LIN {X 0,Y 52.312,Z 344.343,A -85,B 0,C 180,E1 -30110.333,E2 -30110.333} C_VEL
LIN {X 0,Y 48.631,Z 350.268,A -85,B 0,C 180,E1 -30114.672,E2 -30114.672} C_VEL
LIN {X 0,Y 44.07,Z 356.853,A -85,B 0,C 180,E1 -30121.405,E2 -30121.405} C_VEL
LIN {X 0,Y 40.193,Z 362.332,A -85,B 0,C 180,E1 -30129.517,E2 -30129.517} C_VEL
LIN {X 0,Y 37.096,Z 366.924,A -85,B 0,C 180,E1 -30139.065,E2 -30139.065} C_VEL
LIN {X 0,Y 35.067,Z 370.756,A -85,B 0,C 180,E1 -30149.985,E2 -30149.985} C_VEL
LIN {X 0,Y 34.251,Z 375.136,A -85,B 0,C 180,E1 -30167.91,E2 -30167.91} C_VEL
LIN {X 0,Y 36.577,Z 378.214,A -85,B 0,C 180,E1 -30185.182,E2 -30185.182} C_VEL
LIN {X 0,Y 39.68,Z 379.564,A -85,B 0,C 180,E1 -30195.091,E2 -30195.091} C_VEL
LIN {X 0,Y 43.758,Z 380.409,A -85,B 0,C 180,E1 -30203.401,E2 -30203.401} C_VEL
LIN {X 0,Y 48.588,Z 380.746,A -85,B 0,C 180,E1 -30210.19,E2 -30210.19} C_VEL
LIN {X 0,Y 57.076,Z 380.1,A -85,B 0,C 180,E1 -30218.335,E2 -30218.335} C_VEL
LIN {X 0,Y 65.755,Z 378.362,A -85,B 0,C 180,E1 -30224.109,E2 -30224.109} C_VEL
LIN {X 0,Y 71.786,Z 376.474,A -85,B 0,C 180,E1 -30228.719,E2 -30228.719} C_VEL
LIN {X 0,Y 73.199,Z 375.693,A -85,B 0,C 180,E1 -30234.5,E2 -30234.5} C_VEL
LIN {X 0,Y 74.379,Z 375.201,A -85,B 0,C 180,E1 -30240.01,E2 -30240.01} C_VEL
LIN {X 0,Y 74.561,Z 375.241,A -85,B 0,C 180,E1 -30245.418,E2 -30245.418} C_VEL
LIN {X 0,Y 73.493,Z 376.057,A -85,B 0,C 180,E1 -30251.036,E2 -30251.036} C_VEL
LIN {X 0,Y 72.047,Z 377.224,A -85,B 0,C 180,E1 -30257.272,E2 -30257.272} C_VEL
LIN {X 0,Y 70.354,Z 378.704,A -85,B 0,C 180,E1 -30263.562,E2 -30263.562} C_VEL
LIN {X 0,Y 69.513,Z 379.123,A -85,B 0,C 180,E1 -30264.524,E2 -30264.524} C_VEL
LIN {X 0,Y 63.577,Z 380.886,A -85,B 0,C 180,E1 -30267.848,E2 -30267.848} C_VEL
LIN {X 0,Y 53.603,Z 382.795,A -85,B 0,C 180,E1 -30274.935,E2 -30274.935} C_VEL
LIN {X 0,Y 48.77,Z 383.251,A -85,B 0,C 180,E1 -30278.723,E2 -30278.723} C_VEL
LIN {X 0,Y 40.208,Z 383.047,A -85,B 0,C 180,E1 -30285.215,E2 -30285.215} C_VEL
LIN {X 0,Y 32.533,Z 381.802,A -85,B 0,C 180,E1 -30294.985,E2 -30294.985} C_VEL
LIN {X 0,Y 29.534,Z 380.576,A -85,B 0,C 180,E1 -30304.148,E2 -30304.148} C_VEL
LIN {X 0,Y 27.722,Z 378.087,A -85,B 0,C 180,E1 -30322.737,E2 -30322.737} C_VEL
LIN {X 0,Y 27.585,Z 376.948,A -85,B 0,C 180,E1 -30330.019,E2 -30330.019} C_VEL
LIN {X 0,Y 28.695,Z 372.184,A -85,B 0,C 180,E1 -30351.573,E2 -30351.573} C_VEL
LIN {X 0,Y 32.146,Z 366.987,A -85,B 0,C 180,E1 -30366.978,E2 -30366.978} C_VEL
LIN {X 0,Y 36.196,Z 361.884,A -85,B 0,C 180,E1 -30376.75,E2 -30376.75} C_VEL
LIN {X 0,Y 39.562,Z 357.386,A -85,B 0,C 180,E1 -30383.094,E2 -30383.094} C_VEL
LIN {X 0,Y 44.538,Z 349.245,A -85,B 0,C 180,E1 -30391.727,E2 -30391.727} C_VEL
LIN {X 0,Y 46.548,Z 345.588,A -85,B 0,C 180,E1 -30394.972,E2 -30394.972} C_VEL
LIN {X 0,Y 47.318,Z 343.667,A -85,B 0,C 180,E1 -30396.802,E2 -30396.802} C_VEL
LIN {X 0,Y 46.849,Z 341.036,A -85,B 0,C 180,E1 -30402.525,E2 -30402.525} C_VEL
LIN {X 0,Y 46.325,Z 338.011,A -85,B 0,C 180,E1 -30411.258,E2 -30411.258} C_VEL
LIN {X 0,Y 46.238,Z 335.697,A -85,B 0,C 180,E1 -30419.984,E2 -30419.984} C_VEL
LIN {X 0,Y 45.909,Z 335.406,A -85,B 0,C 180,E1 -30428.79,E2 -30428.79} C_VEL
LIN {X 0,Y 45.63,Z 336.738,A -85,B 0,C 180,E1 -30437.924,E2 -30437.924} C_VEL
LIN {X 0,Y 46.049,Z 338.596,A -85,B 0,C 180,E1 -30447.231,E2 -30447.231} C_VEL
LIN {X 0,Y 46.547,Z 342.331,A -85,B 0,C 180,E1 -30457.133,E2 -30457.133} C_VEL
LIN {X 0,Y 46.644,Z 345.23,A -85,B 0,C 180,E1 -30463.167,E2 -30463.167} C_VEL
LIN {X 0,Y 46.525,Z 346.436,A -85,B 0,C 180,E1 -30465.195,E2 -30465.195} C_VEL
LIN {X 0,Y 41.688,Z 353.188,A -85,B 0,C 180,E1 -30470.771,E2 -30470.771} C_VEL
LIN {X 0,Y 35.669,Z 360.78,A -85,B 0,C 180,E1 -30480.473,E2 -30480.473} C_VEL
LIN {X 0,Y 30.066,Z 367.75,A -85,B 0,C 180,E1 -30496.464,E2 -30496.464} C_VEL
LIN {X 0,Y 27.787,Z 371.491,A -85,B 0,C 180,E1 -30509.981,E2 -30509.981} C_VEL
LIN {X 0,Y 27.068,Z 374.57,A -85,B 0,C 180,E1 -30525.029,E2 -30525.029} C_VEL
LIN {X 0,Y 28.132,Z 376.979,A -85,B 0,C 180,E1 -30539.954,E2 -30539.954} C_VEL
LIN {X 0,Y 30.866,Z 378.768,A -85,B 0,C 180,E1 -30553.061,E2 -30553.061} C_VEL
LIN {X 0,Y 34.882,Z 380.032,A -85,B 0,C 180,E1 -30563.674,E2 -30563.674} C_VEL
LIN {X 0,Y 39.817,Z 380.792,A -85,B 0,C 180,E1 -30571.922,E2 -30571.922} C_VEL
LIN {X 0,Y 45.381,Z 381.059,A -85,B 0,C 180,E1 -30578.278,E2 -30578.278} C_VEL
LIN {X 0,Y 53.7,Z 380.478,A -85,B 0,C 180,E1 -30584.84,E2 -30584.84} C_VEL
LIN {X 0,Y 57.643,Z 379.892,A -85,B 0,C 180,E1 -30587.218,E2 -30587.218} C_VEL
LIN {X 0,Y 64.036,Z 378.502,A -85,B 0,C 180,E1 -30590.969,E2 -30590.969} C_VEL
LIN {X 0,Y 66.038,Z 377.986,A -85,B 0,C 180,E1 -30593.902,E2 -30593.902} C_VEL
LIN {X 0,Y 67.498,Z 377.51,A -85,B 0,C 180,E1 -30600.011,E2 -30600.011} C_VEL
LIN {X 0,Y 67.563,Z 377.651,A -85,B 0,C 180,E1 -30605.981,E2 -30605.981} C_VEL
LIN {X 0,Y 66.302,Z 378.498,A -85,B 0,C 180,E1 -30612.25,E2 -30612.25} C_VEL
LIN {X 0,Y 65.571,Z 378.99,A -85,B 0,C 180,E1 -30615.315,E2 -30615.315} C_VEL
LIN {X 0,Y 64.344,Z 379.649,A -85,B 0,C 180,E1 -30619.139,E2 -30619.139} C_VEL
LIN {X 0,Y 60.571,Z 380.75,A -85,B 0,C 180,E1 -30621.864,E2 -30621.864} C_VEL
LIN {X 0,Y 54.378,Z 381.959,A -85,B 0,C 180,E1 -30625.241,E2 -30625.241} C_VEL
LIN {X 0,Y 48.371,Z 382.714,A -85,B 0,C 180,E1 -30629.359,E2 -30629.359} C_VEL
LIN {X 0,Y 42.693,Z 383.027,A -85,B 0,C 180,E1 -30634.628,E2 -30634.628} C_VEL
LIN {X 0,Y 37.627,Z 382.789,A -85,B 0,C 180,E1 -30641.68,E2 -30641.68} C_VEL
LIN {X 0,Y 33.266,Z 382.045,A -85,B 0,C 180,E1 -30650.69,E2 -30650.69} C_VEL
LIN {X 0,Y 29.534,Z 380.576,A -85,B 0,C 180,E1 -30664.148,E2 -30664.148} C_VEL
LIN {X 0,Y 28.094,Z 379.743,A -85,B 0,C 180,E1 -30671.141,E2 -30671.141} C_VEL
LIN {X 0,Y 26.518,Z 378.551,A -85,B 0,C 180,E1 -30678.34,E2 -30678.34} C_VEL
LIN {X 0,Y 23.678,Z 375.861,A -85,B 0,C 180,E1 -30694.212,E2 -30694.212} C_VEL
LIN {X 0,Y 22.692,Z 371.629,A -85,B 0,C 180,E1 -30717.059,E2 -30717.059} C_VEL
LIN {X 0,Y 24.484,Z 368.631,A -85,B 0,C 180,E1 -30729.245,E2 -30729.245} C_VEL
LIN {X 0,Y 30.422,Z 362.298,A -85,B 0,C 180,E1 -30743.984,E2 -30743.984} C_VEL
LIN {X 0,Y 34.332,Z 357.924,A -85,B 0,C 180,E1 -30750.49,E2 -30750.49} C_VEL
LIN {X 0,Y 40.415,Z 349.482,A -85,B 0,C 180,E1 -30759.629,E2 -30759.629} C_VEL
LIN {X 0,Y 41.527,Z 347.732,A -85,B 0,C 180,E1 -30761.161,E2 -30761.161} C_VEL
LIN {X 0,Y 41.968,Z 346.588,A -85,B 0,C 180,E1 -30762.941,E2 -30762.941} C_VEL
LIN {X 0,Y 41.912,Z 344.179,A -85,B 0,C 180,E1 -30770.329,E2 -30770.329} C_VEL
LIN {X 0,Y 41.988,Z 341.773,A -85,B 0,C 180,E1 -30779.983,E2 -30779.983} C_VEL
LIN {X 0,Y 41.698,Z 341.499,A -85,B 0,C 180,E1 -30789.686,E2 -30789.686} C_VEL
LIN {X 0,Y 41.509,Z 343.851,A -85,B 0,C 180,E1 -30804.97,E2 -30804.97} C_VEL
LIN {X 0,Y 41.384,Z 346.403,A -85,B 0,C 180,E1 -30813.472,E2 -30813.472} C_VEL
LIN {X 0,Y 41.277,Z 348.028,A -85,B 0,C 180,E1 -30817.58,E2 -30817.58} C_VEL
LIN {X 0,Y 40.319,Z 349.767,A -85,B 0,C 180,E1 -30819.59,E2 -30819.59} C_VEL
LIN {X 0,Y 33.592,Z 357.534,A -85,B 0,C 180,E1 -30827.139,E2 -30827.139} C_VEL
LIN {X 0,Y 28.386,Z 363.011,A -85,B 0,C 180,E1 -30836.125,E2 -30836.125} C_VEL
LIN {X 0,Y 23.131,Z 368.576,A -85,B 0,C 180,E1 -30852.289,E2 -30852.289} C_VEL
LIN {X 0,Y 20.519,Z 372.222,A -85,B 0,C 180,E1 -30869.974,E2 -30869.974} C_VEL
LIN {X 0,Y 20.827,Z 376.416,A -85,B 0,C 180,E1 -30900.38,E2 -30900.38} C_VEL
LIN {X 0,Y 25.998,Z 379.32,A -85,B 0,C 180,E1 -30924.156,E2 -30924.156} C_VEL
LIN {X 0,Y 31.096,Z 380.5,A -85,B 0,C 180,E1 -30934.653,E2 -30934.653} C_VEL
LIN {X 0,Y 36.928,Z 381.176,A -85,B 0,C 180,E1 -30942.049,E2 -30942.049} C_VEL
LIN {X 0,Y 43.206,Z 381.357,A -85,B 0,C 180,E1 -30947.356,E2 -30947.356} C_VEL
LIN {X 0,Y 51.106,Z 380.855,A -85,B 0,C 180,E1 -30952.11,E2 -30952.11} C_VEL
LIN {X 0,Y 56.454,Z 380.113,A -85,B 0,C 180,E1 -30954.72,E2 -30954.72} C_VEL
LIN {X 0,Y 59.746,Z 379.467,A -85,B 0,C 180,E1 -30957.514,E2 -30957.514} C_VEL
LIN {X 0,Y 60.383,Z 379.35,A -85,B 0,C 180,E1 -30960.012,E2 -30960.012} C_VEL
LIN {X 0,Y 60.338,Z 379.584,A -85,B 0,C 180,E1 -30966.701,E2 -30966.701} C_VEL
LIN {X 0,Y 58.741,Z 380.398,A -85,B 0,C 180,E1 -30973.857,E2 -30973.857} C_VEL
LIN {X 0,Y 58.211,Z 380.609,A -85,B 0,C 180,E1 -30975.049,E2 -30975.049} C_VEL
LIN {X 0,Y 51.742,Z 381.744,A -85,B 0,C 180,E1 -30978.083,E2 -30978.083} C_VEL
LIN {X 0,Y 45.311,Z 382.422,A -85,B 0,C 180,E1 -30981.498,E2 -30981.498} C_VEL
LIN {X 0,Y 39.092,Z 382.661,A -85,B 0,C 180,E1 -30986.018,E2 -30986.018} C_VEL
LIN {X 0,Y 33.325,Z 382.414,A -85,B 0,C 180,E1 -30992.511,E2 -30992.511} C_VEL
LIN {X 0,Y 28.134,Z 381.6,A -85,B 0,C 180,E1 -31001.489,E2 -31001.489} C_VEL
LIN {X 0,Y 23.105,Z 379.897,A -85,B 0,C 180,E1 -31017.795,E2 -31017.795} C_VEL
LIN {X 0,Y 20.712,Z 377.481,A -85,B 0,C 180,E1 -31040.258,E2 -31040.258} C_VEL
LIN {X 0,Y 20.506,Z 376.288,A -85,B 0,C 180,E1 -31050.026,E2 -31050.026} C_VEL
LIN {X 0,Y 21.131,Z 373.245,A -85,B 0,C 180,E1 -31069.452,E2 -31069.452} C_VEL
LIN {X 0,Y 24.484,Z 368.631,A -85,B 0,C 180,E1 -31089.245,E2 -31089.245} C_VEL
LIN {X 0,Y 25.897,Z 366.591,A -85,B 0,C 180,E1 -31096.276,E2 -31096.276} C_VEL
LIN {X 0,Y 27.445,Z 363.067,A -85,B 0,C 180,E1 -31108.065,E2 -31108.065} C_VEL
LIN {X 0,Y 29.567,Z 359.151,A -85,B 0,C 180,E1 -31118.415,E2 -31118.415} C_VEL
LIN {X 0,Y 31.596,Z 356.479,A -85,B 0,C 180,E1 -31122.637,E2 -31122.637} C_VEL
LIN {X 0,Y 36.913,Z 350.079,A -85,B 0,C 180,E1 -31129.004,E2 -31129.004} C_VEL
LIN {X 0,Y 37.338,Z 347.51,A -85,B 0,C 180,E1 -31139.981,E2 -31139.981} C_VEL
LIN {X 0,Y 37.028,Z 347.337,A -85,B 0,C 180,E1 -31150.921,E2 -31150.921} C_VEL
LIN {X 0,Y 36.672,Z 348.833,A -85,B 0,C 180,E1 -31162.516,E2 -31162.516} C_VEL
LIN {X 0,Y 36.182,Z 350.978,A -85,B 0,C 180,E1 -31170.728,E2 -31170.728} C_VEL
LIN {X 0,Y 30.327,Z 357.155,A -85,B 0,C 180,E1 -31175.769,E2 -31175.769} C_VEL
LIN {X 0,Y 22.775,Z 363.947,A -85,B 0,C 180,E1 -31185.997,E2 -31185.997} C_VEL
LIN {X 0,Y 16.383,Z 369.408,A -85,B 0,C 180,E1 -31204.561,E2 -31204.561} C_VEL
LIN {X 0,Y 13.259,Z 372.953,A -85,B 0,C 180,E1 -31229.96,E2 -31229.96} C_VEL
LIN {X 0,Y 14.975,Z 377.058,A -85,B 0,C 180,E1 -31274.696,E2 -31274.696} C_VEL
LIN {X 0,Y 22.507,Z 379.867,A -85,B 0,C 180,E1 -31299.45,E2 -31299.45} C_VEL
LIN {X 0,Y 28.727,Z 380.969,A -85,B 0,C 180,E1 -31308.034,E2 -31308.034} C_VEL
LIN {X 0,Y 35.363,Z 381.559,A -85,B 0,C 180,E1 -31313.425,E2 -31313.425} C_VEL
LIN {X 0,Y 42.211,Z 381.657,A -85,B 0,C 180,E1 -31317.147,E2 -31317.147} C_VEL
LIN {X 0,Y 50.943,Z 381.03,A -85,B 0,C 180,E1 -31320.592,E2 -31320.592} C_VEL
LIN {X 0,Y 53.315,Z 380.742,A -85,B 0,C 180,E1 -31322.178,E2 -31322.178} C_VEL
LIN {X 0,Y 52.817,Z 381.024,A -85,B 0,C 180,E1 -31327.66,E2 -31327.66} C_VEL
LIN {X 0,Y 49.985,Z 381.529,A -85,B 0,C 180,E1 -31330.254,E2 -31330.254} C_VEL
LIN {X 0,Y 43.215,Z 382.131,A -85,B 0,C 180,E1 -31332.695,E2 -31332.695} C_VEL
LIN {X 0,Y 36.537,Z 382.292,A -85,B 0,C 180,E1 -31335.95,E2 -31335.95} C_VEL
LIN {X 0,Y 30.1,Z 382.011,A -85,B 0,C 180,E1 -31340.992,E2 -31340.992} C_VEL
LIN {X 0,Y 24.029,Z 381.154,A -85,B 0,C 180,E1 -31348.712,E2 -31348.712} C_VEL
LIN {X 0,Y 18.646,Z 379.803,A -85,B 0,C 180,E1 -31361.119,E2 -31361.119} C_VEL
LIN {X 0,Y 13.793,Z 376.876,A -85,B 0,C 180,E1 -31395.279,E2 -31395.279} C_VEL
LIN {X 0,Y 13.412,Z 375.596,A -85,B 0,C 180,E1 -31410.039,E2 -31410.039} C_VEL
LIN {X 0,Y 14.616,Z 372.508,A -85,B 0,C 180,E1 -31438.781,E2 -31438.781} C_VEL
LIN {X 0,Y 19.728,Z 367.549,A -85,B 0,C 180,E1 -31463.323,E2 -31463.323} C_VEL
LIN {X 0,Y 26.845,Z 361.276,A -85,B 0,C 180,E1 -31476.438,E2 -31476.438} C_VEL
LIN {X 0,Y 31.596,Z 356.479,A -85,B 0,C 180,E1 -31482.637,E2 -31482.637} C_VEL
LIN {X 0,Y 32.598,Z 354.899,A -85,B 0,C 180,E1 -31485.644,E2 -31485.644} C_VEL
LIN {X 0,Y 32.946,Z 353.552,A -85,B 0,C 180,E1 -31490.747,E2 -31490.747} C_VEL
LIN {X 0,Y 32.769,Z 352.776,A -85,B 0,C 180,E1 -31496.998,E2 -31496.998} C_VEL
LIN {X 0,Y 32.198,Z 352.596,A -85,B 0,C 180,E1 -31506.875,E2 -31506.875} C_VEL
LIN {X 0,Y 31.704,Z 353.267,A -85,B 0,C 180,E1 -31516.859,E2 -31516.859} C_VEL
LIN {X 0,Y 31.65,Z 353.411,A -85,B 0,C 180,E1 -31518.154,E2 -31518.154} C_VEL
LIN {X 0,Y 30.231,Z 355.072,A -85,B 0,C 180,E1 -31521.533,E2 -31521.533} C_VEL
LIN {X 0,Y 21.676,Z 362.474,A -85,B 0,C 180,E1 -31526.866,E2 -31526.866} C_VEL
LIN {X 0,Y 13.383,Z 368.279,A -85,B 0,C 180,E1 -31537.967,E2 -31537.967} C_VEL
LIN {X 0,Y 7.38,Z 372.304,A -85,B 0,C 180,E1 -31565.166,E2 -31565.166} C_VEL
LIN {X 0,Y 8.193,Z 376.496,A -85,B 0,C 180,E1 -31648.946,E2 -31648.946} C_VEL
LIN {X 0,Y 14.251,Z 378.717,A -85,B 0,C 180,E1 -31670.281,E2 -31670.281} C_VEL
LIN {X 0,Y 23.114,Z 380.697,A -85,B 0,C 180,E1 -31680.031,E2 -31680.031} C_VEL
LIN {X 0,Y 32.413,Z 381.79,A -85,B 0,C 180,E1 -31684.464,E2 -31684.464} C_VEL
LIN {X 0,Y 28.34,Z 381.579,A -85,B 0,C 180,E1 -31687.42,E2 -31687.42} C_VEL
LIN {X 0,Y 21.536,Z 380.707,A -85,B 0,C 180,E1 -31691.883,E2 -31691.883} C_VEL
LIN {X 0,Y 14.966,Z 379.278,A -85,B 0,C 180,E1 -31700.191,E2 -31700.191} C_VEL
LIN {X 0,Y 7.192,Z 376.273,A -85,B 0,C 180,E1 -31740.834,E2 -31740.834} C_VEL
LIN {X 0,Y 6.989,Z 373.382,A -85,B 0,C 180,E1 -31800.271,E2 -31800.271} C_VEL
LIN {X 0,Y 14.881,Z 367.818,A -85,B 0,C 180,E1 -31840.942,E2 -31840.942} C_VEL
LIN {X 0,Y 23.168,Z 361.69,A -85,B 0,C 180,E1 -31850.501,E2 -31850.501} C_VEL
LIN {X 0,Y 28.509,Z 357.025,A -85,B 0,C 180,E1 -31854.821,E2 -31854.821} C_VEL
LIN {X 0,Y 31.151,Z 354.307,A -85,B 0,C 180,E1 -31856.972,E2 -31856.972} C_VEL
LIN {X 0,Y 32.244,Z 352.955,A -85,B 0,C 180,E1 -31859.978,E2 -31859.978} C_VEL
LIN {X 0,Y 31.939,Z 352.852,A -85,B 0,C 180,E1 -31872.688,E2 -31872.688} C_VEL
LIN {X 0,Y 31.704,Z 353.267,A -85,B 0,C 180,E1 -31876.859,E2 -31876.859} C_VEL
LIN {X 0,Y 31.606,Z 355.229,A -85,B 0,C 180,E1 -31879.766,E2 -31879.766} C_VEL
LIN {X 0,Y 31.606,Z 600,A -85,B 0,C 180,E1 -31879.766,E2 -31879.766} C_VEL
LIN {X 0,Y 31.606,Z 600,A -85,B 0,C 180,E1 -31879.766,E2 -31879.766}

QRS_NEXT_CUT()

QRS_NEXT()
QRS_HOME()

END
